TYPE ST_BWK_Stellwert :
STRUCT
	Betrieb		: BOOL;
	Freigabe	: BOOL;
	Modus		: SINT;
	Leistung	: SINT;
	Temperatur	: REAL;
END_STRUCT
END_TYPE

(* stored: Version 1.1.0.1, ProductVersion 3.1.4024.9
   DUT ST_BWK_Stellwert: Id {1c162384-87e7-4488-b4b0-da2cce903aa0} *)
